// TIA Portal V20 export
DATA_BLOCK "instAlarmCounter1"   // DB37
// stored: InstanceOfName LER_AlarmCounter, InstanceOfType FB
"LER_AlarmCounter"
   // VAR_INPUT
   //    productionMode : Bool;
   //    countUp : Bool;
   //    countReset : Bool;
   // END_VAR
   // VAR_IN_OUT
   //    hmiInterface : "LER_typeAlarmCounterInterface";
   // END_VAR
   // VAR
   //    statPulse_Up : Bool;
   //    statPulse_Reset : Bool;
   //    statTonTimer : TON_TIME;
   // END_VAR
BEGIN
END_DATA_BLOCK
